{attribute 'GeneratedUsingTerminal: EK1100-0000-0018'}
{attribute addProperty BoxType "EK1100-0000-0018"}
{attribute addProperty Id "Beckhoff_CUxxxxEK1122Beckhoff_CUxxxxEK1122_BE344318126"}
{attribute addProperty CRC "3920467250"}
{attribute addProperty Size "126"}
TYPE Beckhoff_CUxxxx_E9AD9532 EXTENDS EK1100_1FC0878B :
STRUCT
	{attribute addProperty Name "Beckhoff CUxxxxEK1122"}
	{attribute addProperty PreviousPort "Beckhoff CUxxxx : B"}
	Beckhoff_CUxxxxEK1122 : Beckhoff_CUxxxxEK1122_BE344318;
END_STRUCT
END_TYPE

(* stored: Version 1.2.0.0, ProductVersion 3.1.4024.9
   DUT Beckhoff_CUxxxx_E9AD9532: Id {0fa16d32-d7e9-43ad-997a-1f3afed6fb18} *)
